{attribute 'qualified_only'}
{attribute 'strict'}
{attribute 'to_string'}
TYPE E_FilterMaterial :
(
    Silicon := 0,
    Diamond,
    Germanium
);
END_TYPE

(* stored: Version 1.1.0.1
   DUT E_FilterMaterial: Id {536c2724-7ec8-40a6-b624-2ad540293c94} *)
